{attribute 'qualified_only'}
VAR_GLOBAL
	

END_VAR

(* stored: Version 1.1.0.1, ProductVersion 3.1.4024.15
   GVL GVL: Id {f87f5863-ef76-4681-aea0-d4e152a15836} *)
